// TIA Portal V17 export
// export: Created 2023-12-22T15:04:39.6410723Z, ExportSetting WithDefaults, DisplayName Totally Integrated Automation Portal, DisplayVersion V17, DisplayName TIA Portal Openness, DisplayVersion V17, DisplayName TIA Portal Version Control Interface, DisplayVersion V17, DisplayName STEP 7 Professional, DisplayVersion V17, DisplayName STEP 7 Safety, DisplayVersion V17, DisplayName WinCC Advanced, DisplayVersion V17
FUNCTION_BLOCK "Main_Logick"   // FB1, LAD
{ S7_Optimized_Access := 'FALSE' }
VERSION : 0.1
// stored: AutoNumber true, IsIECCheckEnabled false, SetENOAutomatically false, UDAEnableTagReadback false
   VAR DB_SPECIFIC
      Start : Bool;   // Запуск установки
      Start_Local : Bool;
      REQ_Pump : Bool;   // Запрос запуска насоса
      ev : Bool;
      Ready : Bool;   // Установка готова к работе
      Local : Bool;   // 0-местный, 1-дистанционный
      Mode : Bool;   // 0 - Работа по Гц, 1 - Работа по RM
      SP_Pump { S7_SetPoint := 'True'} : Real;   // уставка для работы по Гц
      RM : Real;   // Расходомер (получаем по MoodBus)
      RM_SP { S7_SetPoint := 'True'} : Real;   // Уставка расхода для насоса
      Level_Norm { S7_SetPoint := 'True'} : Real := 50.0;   // Рабочая точка насоса по уровню
      Distance { S7_SetPoint := 'True'} : Real := 500.0;   // Расстояние от ЩКД1 до скважины
      LE_Bar : Real;   // Показания датчика уровня на панели
      LE_Skvaz { S7_SetPoint := 'True'} : Real := 100.0;   // Глубина скважины
      LE_Skvaz_RCHV { S7_SetPoint := 'True'} : Real;   // Высота скважины относительно резервуара (для рассчета эфективности)
      Effect : Real;   // Эфективность скважины
      Alarm : Word;   // Слово аварий
      Alarms : Struct   // Список аварий
         Leak : Bool;   // Протечка
         Level_Norm : Bool;   // Уровень не в норме
         LE_Warning : Bool;   // Уровень ниже рабочей точки (Предупреждение)
         LE_Alarm : Bool;   // Уровень в аварийной зоне
      END_STRUCT;
   END_VAR
   VAR
      PID_Pump { S7_SetPoint := 'True'} : "PID_ex";   // ПИД Насоса
   END_VAR
   VAR_TEMP   // added for the SCL form of the ladder/FBD networks
      _w1 : Bool;
      _w2 : Bool;
      _w3 : Bool;
      _w4 : Bool;
   END_VAR
BEGIN

REGION Network 1: Готовность скважины к работе
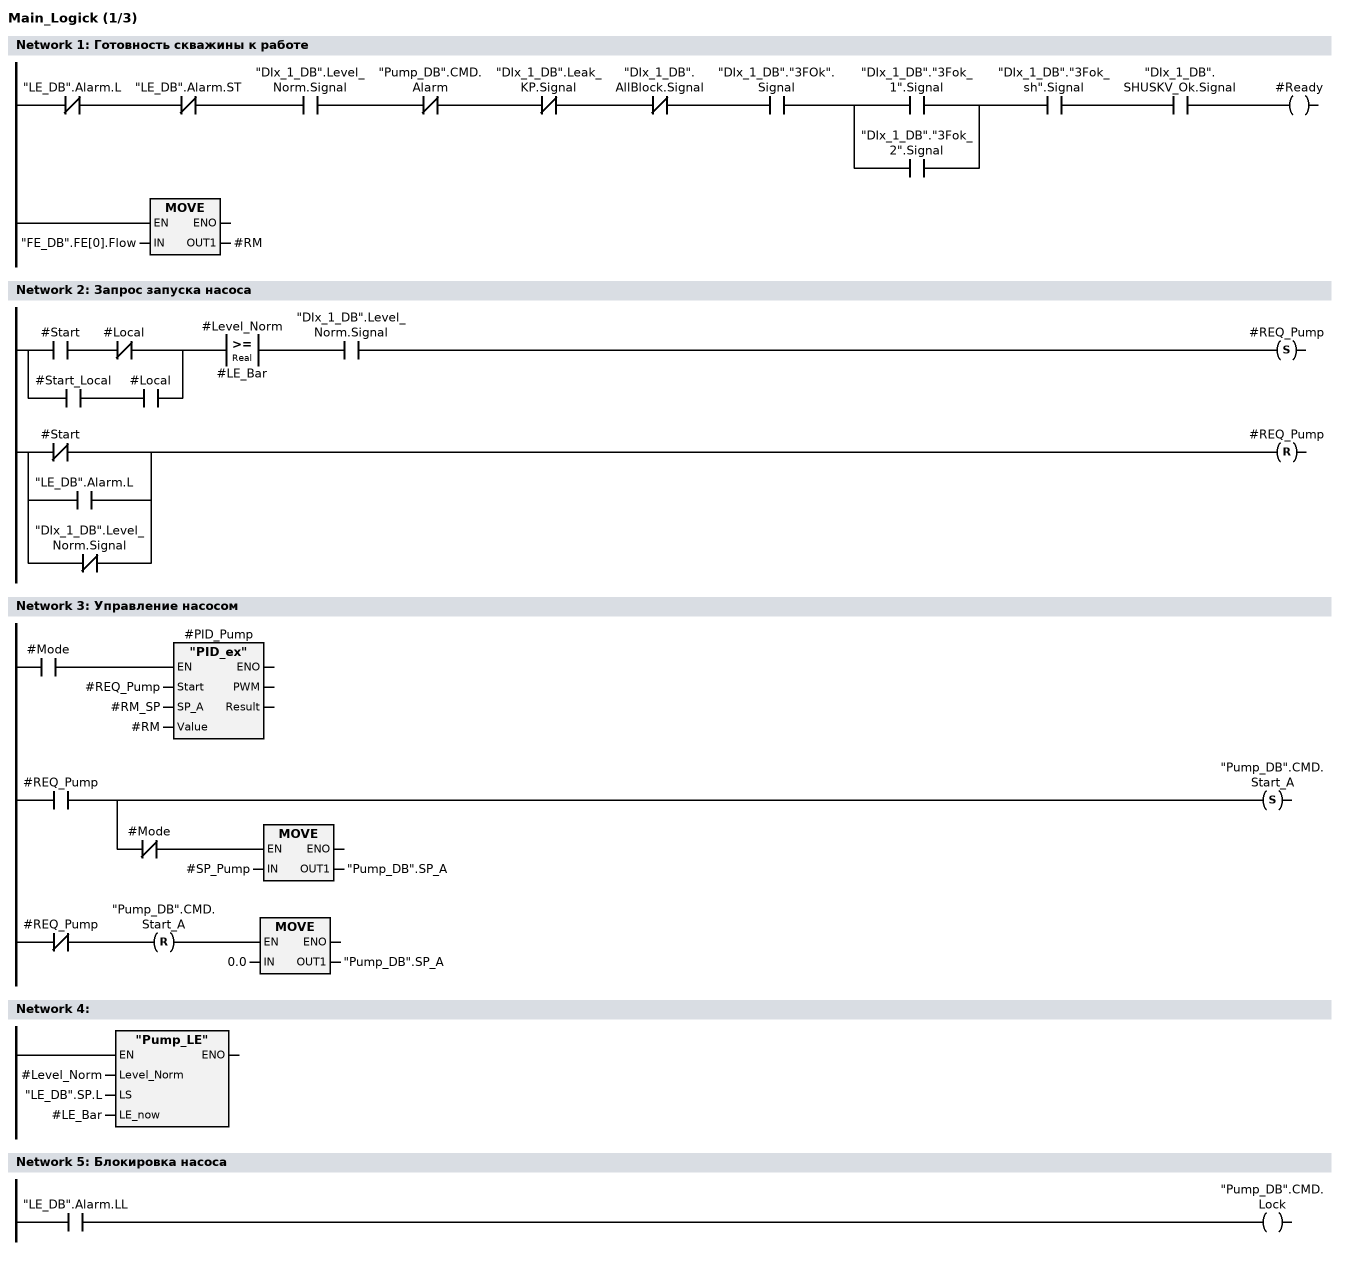
   RUNG wire#powerrail
      I_Contact( "LE_DB".Alarm.L )
      I_Contact( "LE_DB".Alarm.ST )
      Contact( "DIx_1_DB".Level_Norm.Signal )
      I_Contact( "Pump_DB".CMD.Alarm )
      I_Contact( "DIx_1_DB".Leak_KP.Signal )
      I_Contact( "DIx_1_DB".AllBlock.Signal )
      Contact( "DIx_1_DB"."3FOk".Signal )
      wire#w1
      Contact( "DIx_1_DB"."3Fok_1".Signal )
      wire#w2
      Contact( "DIx_1_DB"."3Fok_sh".Signal )
      Contact( "DIx_1_DB".SHUSKV_Ok.Signal )
      Coil( #Ready )
   END_RUNG
   RUNG wire#w1
      Contact( "DIx_1_DB"."3Fok_2".Signal )
   END_RUNG wire#w2
   RUNG wire#powerrail
      Move(in := "FE_DB".FE[0].Flow, out1 => #RM)
   END_RUNG
   // the same network as SCL:
   #Ready := NOT "LE_DB".Alarm.L AND NOT "LE_DB".Alarm.ST AND "DIx_1_DB".Level_Norm.Signal AND NOT "Pump_DB".CMD.Alarm AND NOT "DIx_1_DB".Leak_KP.Signal AND NOT "DIx_1_DB".AllBlock.Signal AND "DIx_1_DB"."3FOk".Signal AND ("DIx_1_DB"."3Fok_1".Signal OR "DIx_1_DB"."3Fok_2".Signal) AND "DIx_1_DB"."3Fok_sh".Signal AND "DIx_1_DB".SHUSKV_Ok.Signal;
   #RM := "FE_DB".FE[0].Flow;
END_REGION

REGION Network 2: Запрос запуска насоса
   RUNG wire#powerrail
      Contact( #Start )
      I_Contact( #Local )
      wire#w1
      { S7_Templates := "SrcType := Real" } GE_Contact(in1 := #Level_Norm, in2 := #LE_Bar)
      Contact( "DIx_1_DB".Level_Norm.Signal )
      S_Coil( #REQ_Pump )
   END_RUNG
   RUNG wire#powerrail
      Contact( #Start_Local )
      Contact( #Local )
   END_RUNG wire#w1
   RUNG wire#powerrail
      I_Contact( #Start )
      wire#w2
      R_Coil( #REQ_Pump )
   END_RUNG
   RUNG wire#powerrail
      Contact( "LE_DB".Alarm.L )
   END_RUNG wire#w2
   RUNG wire#powerrail
      I_Contact( "DIx_1_DB".Level_Norm.Signal )
   END_RUNG wire#w2
   // the same network as SCL:
   IF ((#Start AND NOT #Local) OR (#Start_Local AND #Local)) AND (#Level_Norm >= #LE_Bar) AND "DIx_1_DB".Level_Norm.Signal THEN
       #REQ_Pump := TRUE;
   END_IF;
   IF NOT #Start OR "LE_DB".Alarm.L OR NOT "DIx_1_DB".Level_Norm.Signal THEN #REQ_Pump := FALSE; END_IF;
END_REGION

REGION Network 3: Управление насосом
   RUNG wire#powerrail
      Contact( #Mode )
      #PID_Pump(Start := #REQ_Pump, SP_A := #RM_SP, Value := #RM, PWM =>, Result =>)
   END_RUNG
   RUNG wire#powerrail
      Contact( #REQ_Pump )
      wire#w1
      S_Coil( "Pump_DB".CMD.Start_A )
   END_RUNG
   RUNG wire#w1
      I_Contact( #Mode )
      Move(in := #SP_Pump, out1 => "Pump_DB".SP_A)
   END_RUNG
   RUNG wire#powerrail
      I_Contact( #REQ_Pump )
      R_Coil( "Pump_DB".CMD.Start_A )
      Move(in := 0.0, out1 => "Pump_DB".SP_A)
   END_RUNG
   // the same network as SCL:
   IF #Mode THEN
       #PID_Pump(Start := #REQ_Pump, SP_A := #RM_SP, Value := #RM);   // "PID_ex"
   END_IF;
   IF #REQ_Pump THEN "Pump_DB".CMD.Start_A := TRUE; END_IF;
   IF #REQ_Pump AND NOT #Mode THEN "Pump_DB".SP_A := #SP_Pump; END_IF;
   IF NOT #REQ_Pump THEN
       "Pump_DB".CMD.Start_A := FALSE;
       "Pump_DB".SP_A := 0.0;
   END_IF;
END_REGION

REGION Network 4
   RUNG wire#powerrail
      "Pump_LE"(Level_Norm := #Level_Norm, LS := "LE_DB".SP.L, LE_now := #LE_Bar)
   END_RUNG
   // the same network as SCL:
   "Pump_LE"(Level_Norm := #Level_Norm, LS := "LE_DB".SP.L, LE_now := #LE_Bar);
END_REGION

REGION Network 5: Блокировка насоса
   RUNG wire#powerrail
      Contact( "LE_DB".Alarm.LL )
      Coil( "Pump_DB".CMD.Lock )
   END_RUNG
   // the same network as SCL:
   "Pump_DB".CMD.Lock := "LE_DB".Alarm.LL;
END_REGION

REGION Network 6: Датчики перелива и уровня (Аварии)
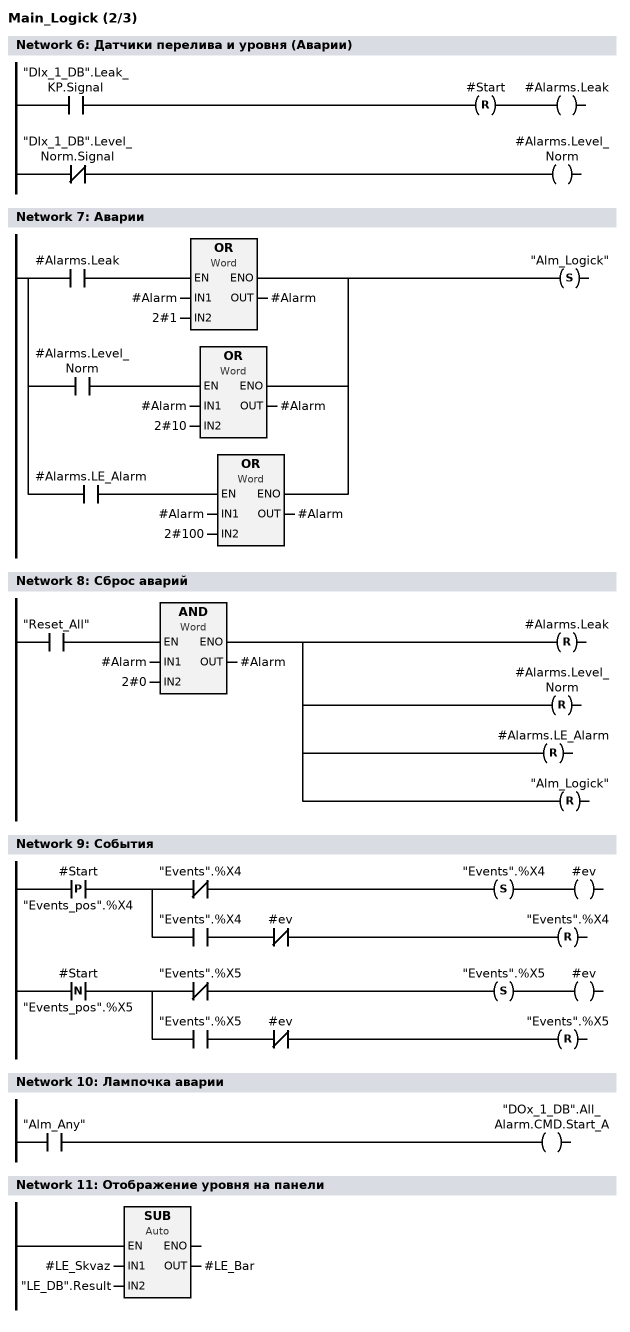
   RUNG wire#powerrail
      Contact( "DIx_1_DB".Leak_KP.Signal )
      R_Coil( #Start )
      Coil( #Alarms.Leak )
   END_RUNG
   RUNG wire#powerrail
      I_Contact( "DIx_1_DB".Level_Norm.Signal )
      Coil( #Alarms.Level_Norm )
   END_RUNG
   // the same network as SCL:
   IF "DIx_1_DB".Leak_KP.Signal THEN #Start := FALSE; END_IF;
   #Alarms.Leak := "DIx_1_DB".Leak_KP.Signal;
   #Alarms.Level_Norm := NOT "DIx_1_DB".Level_Norm.Signal;
END_REGION

REGION Network 7: Аварии
   IF #Alarms.Leak THEN #Alarm := #Alarm OR 2#1; END_IF;
   IF #Alarms.Level_Norm THEN #Alarm := #Alarm OR 2#10; END_IF;
   IF #Alarms.LE_Alarm THEN #Alarm := #Alarm OR 2#100; END_IF;
   IF #Alarms.Leak OR #Alarms.Level_Norm OR #Alarms.LE_Alarm THEN "Alm_Logick" := TRUE; END_IF;
END_REGION

REGION Network 8: Сброс аварий
   RUNG wire#powerrail
      Contact( "Reset_All" )
      { S7_Templates := "SrcType := Word"; S7_GenerateENO := "TRUE" } And(in1 := #Alarm, in2 := 2#0, out => #Alarm)
      wire#w1
      R_Coil( #Alarms.Leak )
   END_RUNG
   RUNG wire#w1
      R_Coil( #Alarms.Level_Norm )
   END_RUNG
   RUNG wire#w1
      R_Coil( #Alarms.LE_Alarm )
   END_RUNG
   RUNG wire#w1
      R_Coil( "Alm_Logick" )
   END_RUNG
   // the same network as SCL:
   IF "Reset_All" THEN
       #Alarm := #Alarm AND 2#0;
       #Alarms.Leak := FALSE;
       #Alarms.Level_Norm := FALSE;
       #Alarms.LE_Alarm := FALSE;
       "Alm_Logick" := FALSE;
   END_IF;
END_REGION

REGION Network 9: События
   RUNG wire#powerrail
      P_Contact(operand := #Start, bit := "Events_pos".%X4)
      wire#w1
      I_Contact( "Events".%X4 )
      S_Coil( "Events".%X4 )
      Coil( #ev )
   END_RUNG
   RUNG wire#w1
      Contact( "Events".%X4 )
      I_Contact( #ev )
      R_Coil( "Events".%X4 )
   END_RUNG
   RUNG wire#powerrail
      N_Contact(operand := #Start, bit := "Events_pos".%X5)
      wire#w2
      I_Contact( "Events".%X5 )
      S_Coil( "Events".%X5 )
      Coil( #ev )
   END_RUNG
   RUNG wire#w2
      Contact( "Events".%X5 )
      I_Contact( #ev )
      R_Coil( "Events".%X5 )
   END_RUNG
   // the same network as SCL:
   #_w1 := #Start AND NOT "Events_pos".%X4;   // rising edge of #Start
   "Events_pos".%X4 := #Start;
   #_w2 := #_w1 AND NOT "Events".%X4;
   IF #_w2 THEN "Events".%X4 := TRUE; END_IF;
   #ev := #_w2;
   IF #_w1 AND "Events".%X4 AND NOT #ev THEN "Events".%X4 := FALSE; END_IF;
   #_w3 := NOT #Start AND "Events_pos".%X5;   // falling edge of #Start
   "Events_pos".%X5 := #Start;
   #_w4 := #_w3 AND NOT "Events".%X5;
   IF #_w4 THEN "Events".%X5 := TRUE; END_IF;
   #ev := #_w4;
   IF #_w3 AND "Events".%X5 AND NOT #ev THEN "Events".%X5 := FALSE; END_IF;
END_REGION

REGION Network 10: Лампочка аварии
   RUNG wire#powerrail
      Contact( "Alm_Any" )
      Coil( "DOx_1_DB".All_Alarm.CMD.Start_A )
   END_RUNG
   // the same network as SCL:
   "DOx_1_DB".All_Alarm.CMD.Start_A := "Alm_Any";
END_REGION

REGION Network 11: Отображение уровня на панели
   RUNG wire#powerrail
      Sub(in1 := #LE_Skvaz, in2 := "LE_DB".Result, out => #LE_Bar)
   END_RUNG
   // the same network as SCL:
   #LE_Bar := #LE_Skvaz - "LE_DB".Result;
END_REGION

REGION Network 12: Рассчет эффективности скважины
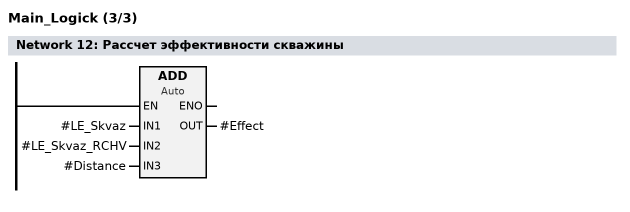
   RUNG wire#powerrail
      Add(in1 := #LE_Skvaz, in2 := #LE_Skvaz_RCHV, in3 := #Distance, out => #Effect)
   END_RUNG
   // the same network as SCL:
   #Effect := #LE_Skvaz + #LE_Skvaz_RCHV + #Distance;
END_REGION
END_FUNCTION_BLOCK
